(* IEC 61131-3 sources: plcassist-cli/packages/volt-cli/test/Volt.Engine.Tests/fixtures/st-fixed-point, 9 files *)

(* ---- block-comment-with-a-blank-line-above-a-member.itf ---- *)
// Modules that react to EStop and Stop events from the machine
INTERFACE IModuleBase
EXTENDS IAbleToRegister, __SYSTEM.IQueryInterface

(* Command to reset the module in case of E-Stop

Add code here to handle emergency stops. For example:

// Reset the state of the unit.
State := MyUnit_State.None;

 *)
METHOD PUBLIC EStop : BOOL	// Returns true when drives are in standstill
END_METHOD

// Command to stop a module
METHOD PUBLIC Stop : BOOL
END_METHOD

END_INTERFACE

(* ---- two-blank-lines-before-body.fun ---- *)
// This function rounds a real down to n digits behind the comma.
FUNCTION Round : REAL
VAR_INPUT
	in	: REAL;
END_VAR
VAR
	X	: REAL;
END_VAR

(*
version 1.5	25. oct. 2008
*)
X := in;
Round := X;

END_FUNCTION

(* ---- wrapped-return-type-no-var-section.fun ---- *)
// Doubles a real. No VAR section, so the wrapped return type is all there is to find.
FUNCTION Compute
: REAL

Compute := 2.0;

END_FUNCTION

(* ---- action-with-a-leading-comment.fb ---- *)
FUNCTION_BLOCK Machine
VAR
	step	: INT;
END_VAR

;

END_FUNCTION_BLOCK

ACTION Reset
// Put every axis back to its home position before the next batch.
step := 0;
END_ACTION

(* ---- property-accessor-with-an-empty-var-block.fb ---- *)
FUNCTION_BLOCK DrawerMagazineFB
VAR
	active	: IDrawer;
END_VAR

;

END_FUNCTION_BLOCK

PROPERTY ActiveDrawerItf : IDrawer
%FOLDER Properties
GET
VAR
END_VAR

// Determine the active and inactive drawer
ActiveDrawerItf := active;
END_GET
END_PROPERTY

(* ---- trailing-space-on-a-boundary-line.fb ---- *)
FUNCTION_BLOCK VirtualMaster
VAR
	MaxTorque	: REAL;
END_VAR

//Max torque on the axis. If the machine does not stop, this keeps the torque sane.
MaxTorque := 100.0;

END_FUNCTION_BLOCK

METHOD PUBLIC Selection
//Selection of the cam.
MaxTorque := 0;
END_METHOD

(* ---- wrapped-header-no-var-section.fb ---- *)
// Control a single output. The output is inverted
{attribute 'symbol' := 'none'}
FUNCTION_BLOCK PUBLIC Cylinder_52Valve_InvertedFB
EXTENDS Cylinder_52ValveFB
IMPLEMENTS IActuator

// Execute base cylinder fb
SUPER^();

END_FUNCTION_BLOCK

METHOD PROTECTED Alarms
// Set the alarm messages (inverted)
SetSensorOutAlarm(inputIn XOR NOT Output.Map());
END_METHOD

(* ---- blank-under-a-members-opening-comment.prg ---- *)
PROGRAM ErrorHandling
VAR
	dummy	: BOOL;
END_VAR

END_PROGRAM

METHOD PROTECTED Initialize
// Connect Lenze module handlers to this base module handler

GlobalVars.fbModuleManager.ModuleHandler.SetParent(
	ModuleHandlerParent	:= ModuleHandler);
END_METHOD

(* ---- member-comment-after-end-var.prg ---- *)
// Helper functions to set or reset bits in integers
{attribute 'hide_all_locals'}
PROGRAM BitLogic
VAR
	uInput		: PointerSizesUnion;
END_VAR

END_PROGRAM

// Population count: Count the number of bits that are 1 in a byte
METHOD PUBLIC CountByte : USINT
VAR_INPUT
	in	: BYTE;			// Count number of 1's
END_VAR

// This method uses Brian Kernighan's algorithm. Google it for more info.
WHILE in <> 0 DO
	CountByte	:= CountByte + 1;
END_WHILE
END_METHOD
